FUNCTION_BLOCK FB_HighVoltTray EXTENDS FB_ActiveTarget

VAR
	//Hardware-Verküpfung
	pHighVoltSupplyRef	: POINTER TO FB_HighVoltSupply;
	
	//Prozessdaten
	nVoltageActual		: DINT;
	nCurrentActual		: DINT;	//in 10tel µA (10 enstpr. 1.0µA)

	//Variablen allgemeine Statemachine
	
	bCurrentMonitoring		: BOOL;
	bPwrCutOffTriggered		: BOOL;

	//Spec-Properties
	nVoltageChannel			: USINT;
	nCurrentLimit			: UINT; 		//Strombegrenzung der HV-Quelle //in 10tel µA (10 enstpr. 1.0µA)
	
	nPowerCutOffThreshold	: UINT;			//Stromüberwachung (Automatisches Abschalten bei Erreichen) //in 10tel µA (10 enstpr. 1.0µA)
											//wenn "0" , dann wird nicht überwacht
	tPowerCutOffTime		: TIME; 		//wenn Strom für diese Zeit die Abschaltschwelle überschreitet, dann wird abgeschaltet
	
	//****************************************Aktionvariablen****************************************************
	
	//Action: "SetVoltage"
	nVoltageSetpoint	: USINT;
	
	//Action: "SetCurrent"
	nCurrentSetpoint	: USINT;
	
	//Action: "SwitchVoltage"
	bVoltageOn			: BOOL;
	
	timer : TON;	//Stromüberwachung
	
	
END_VAR

IF pHighVoltSupplyRef = 0 THEN
	RETURN;
END_IF

pFbSafety^.M_MesBoxOn();

//durch Notaus oder Unlock werden die Kanäle ausgeschalten und müssen in jedem Fall
//manuell durch SwitchVoltage wieder eingeschalten werden
IF NOT pHighVoltSupplyRef^.bHVPSAvailable THEN
	pHighVoltSupplyRef^.M_SwitchVoltage(1,FALSE);
	pHighVoltSupplyRef^.M_SwitchVoltage(2,FALSE);
END_IF

//Stromüberwachung
nCurrentActual := pHighVoltSupplyRef^.M_GetCurrent();
IF bCurrentMonitoring AND NOT bPwrCutOffTriggered THEN
	IF nCurrentActual >= nPowerCutOffThreshold THEN
		//Strom muss für eine vorgegebene Zeit die Abschaltschwelle erreicht haben.
		timer(IN:= TRUE, PT:= tPowerCutOffTime);
		IF timer.Q THEN
			timer(IN:= FALSE);
			bPwrCutOffTriggered := TRUE; 
			pHighVoltSupplyRef^.M_SwitchVoltage(1,FALSE);
			pHighVoltSupplyRef^.M_SwitchVoltage(2,FALSE);
			stError.POU := E_POU.POU_FB_HighVoltTray;
			stError.ErrorId := E_ErrorIdCmd.ERRORID_OverCurrentHighVoltTray;
			stError.ObjectId := nObjectID;
			fbErrorList.M_Add(stError);			
		END_IF
	ELSE
		timer(IN:= FALSE);
	END_IF
END_IF

//Prozessdaten aktualisieren
stProcessData.nObjId := nObjectID;
stProcessData.n32Data[0] := BOOL_TO_DINT(bIsInit);
stProcessData.n32Data[1] := eCurrentState;
stProcessData.n32Data[2] := stError.ErrorId;

IF nVoltageChannel = 1 THEN
	stProcessData.n32Data[3] := BOOL_TO_DINT(NOT pHighVoltSupplyRef^.bDigiOutVoltage1);
ELSIF nVoltageChannel = 2 THEN
	stProcessData.n32Data[3] := BOOL_TO_DINT(NOT pHighVoltSupplyRef^.bDigiOutVoltage2);
END_IF

nVoltageActual := pHighVoltSupplyRef^.M_GetVoltage();
stProcessData.n32Data[4] := nVoltageActual;
stProcessData.n32Data[5] := nCurrentActual;

aObjProcData[nNotifyId] := stProcessData;

METHOD FB_init : BOOL
VAR_INPUT
	bInitRetains : BOOL; // if TRUE, the retain variables are initialized (warm start / cold start)
	bInCopyCode : BOOL;  // if TRUE, the instance afterwards gets moved into the copy code (online change)
END_VAR
eObjectType := E_ObjectType.OBJECTTYPE_HighVoltTray;
eObjectGroup := E_ObjectGroup.OBJECTGROUP_Target OR E_ObjectGroup.OBJECTGROUP_Device;
END_METHOD

METHOD M_CheckProcDataType : BOOL
VAR_INPUT
	eProcDataType : E_ProcDataType;
END_VAR
IF eProcDataType = E_ProcDataType.PROCDATATYPE_Voltage1 OR eProcDataType = E_ProcDataType.PROCDATATYPE_Current1 THEN
	M_CheckProcDataType := TRUE;
END_IF
END_METHOD

METHOD M_CurrentMonitoring
VAR_INPUT
	bOn : BOOL;
END_VAR
IF bOn THEN
	IF nPowerCutOffThreshold > 0 THEN
		bCurrentMonitoring := TRUE;		
	END_IF
ELSE
	bCurrentMonitoring := FALSE;
 	bPwrCutOffTriggered := FALSE;
END_IF
END_METHOD

METHOD M_ExeAction : ERRORID
VAR_INPUT
	refActionData	: REFERENCE TO ST_ActionData;	
END_VAR
CASE refActionData.eAction OF
	E_Action.ACTION_Init:
		bIsInit := TRUE;
		RETURN;
	E_Action.ACTION_SetVoltage:
		IF 	pHighVoltSupplyRef > 0 THEN
			pHighVoltSupplyRef^.M_SetVoltage(DINT_TO_INT(refActionData.aParams[1]));
			pHighVoltSupplyRef^.M_SetCurrent(nCurrentLimit);
		END_IF
	E_Action.ACTION_SwitchVoltage:
		IF 	pHighVoltSupplyRef > 0 THEN
			IF pHighVoltSupplyRef^.bHVPSAvailable THEN
				pHighVoltSupplyRef^.M_SwitchVoltage(nVoltageChannel,DINT_TO_BOOL(refActionData.aParams[1]));
			ELSE
				M_ExeAction := E_ErrorIdCmd.ERRORID_HighVoltSupplyOff;
			END_IF
		ELSE
			M_ExeAction := E_ErrorIdObjMgmt.ERRORID_InvalidHardwareRef;
		END_IF
	ELSE
		M_ExeAction := E_ErrorIdCmd.ERRORID_InvalidAction;	
END_CASE
END_METHOD

METHOD M_GetActionBusy : BOOL
VAR_INPUT
	eAction : E_Action;
END_VAR
IF eAction = eCurrentAction THEN
	M_GetActionBusy := TRUE;
END_IF
END_METHOD

METHOD M_GetAllProps : ERRORID
VAR_INPUT
	refCmdData : REFERENCE TO  ST_CmdData;
END_VAR
SUPER^.M_GetAllProps(refCmdData);
nCurrentPropIndex := nCurrentPropIndex + 1;
refCmdData.n32Data[nCurrentPropIndex] := nVoltageChannel;
nCurrentPropIndex := nCurrentPropIndex + 1;
refCmdData.n32Data[nCurrentPropIndex] := nCurrentLimit;
nCurrentPropIndex := nCurrentPropIndex + 1;
refCmdData.n32Data[nCurrentPropIndex] := nPowerCutOffThreshold;
nCurrentPropIndex := nCurrentPropIndex + 1;
refCmdData.n32Data[nCurrentPropIndex] := TIME_TO_DINT(tPowerCutOffTime);
END_METHOD

METHOD M_GetProcData : DINT
VAR_INPUT
	eProcDataType : E_ProcDataType;
END_VAR
IF eProcDataType = E_ProcDataType.PROCDATATYPE_Voltage1 THEN
	M_GetProcData := pHighVoltSupplyRef^.M_GetVoltage();
ELSIF eProcDataType = E_ProcDataType.PROCDATATYPE_Current1 THEN
	M_GetProcData := pHighVoltSupplyRef^.M_GetCurrent();
END_IF
END_METHOD

METHOD M_Reset
bBusy := TRUE;
eCurrentState := E_MachineState.MACHINESTATE_Reset;
M_CurrentMonitoring(FALSE);
END_METHOD

METHOD M_SetAllProps : ERRORID
VAR_INPUT
	refCmdData : REFERENCE TO  ST_CmdData;
END_VAR
M_SetAllProps := SUPER^.M_SetAllProps(refCmdData);

IF M_SetAllProps > 0 THEN
	RETURN;
END_IF

{IF defined (variable:fbHighVoltSupplyRef)}
pHighVoltSupplyRef := ADR(fbHighVoltSupplyRef);
{ELSE}
{warning 'implement errorId}
M_SetAllProps := E_ErrorIdObjMgmt.ERRORID_InvalidHardwareRef;
{END_IF}
nCurrentPropIndex := nCurrentPropIndex + 1;
nSpecPropIndex := nCurrentPropIndex;
IF refCmdData.n32Data[nCurrentPropIndex] >= 1 AND refCmdData.n32Data[nCurrentPropIndex] <= 2 THEN
	nVoltageChannel := DINT_TO_USINT(refCmdData.n32Data[nCurrentPropIndex]);
ELSE
	M_SetAllProps := E_ErrorIdObjMgmt.ERRORID_InvalidHardwareRef;
END_IF

nCurrentPropIndex := nCurrentPropIndex + 1;
nCurrentLimit := DINT_TO_UINT(refCmdData.n32Data[nCurrentPropIndex]);
nCurrentPropIndex := nCurrentPropIndex + 1;
nPowerCutOffThreshold := DINT_TO_UINT(refCmdData.n32Data[nCurrentPropIndex]);
nCurrentPropIndex := nCurrentPropIndex + 1;
tPowerCutOffTime := DINT_TO_TIME(refCmdData.n32Data[nCurrentPropIndex]);

nNoOfProps := nCurrentPropIndex + 1;
END_METHOD

METHOD M_SetSingleProp : ERRORID
VAR_INPUT
	refCmdData : REFERENCE TO  ST_CmdData;
END_VAR
IF nSpecPropIndex = refCmdData.aHeader[1] THEN
	IF refCmdData.n32Data[0] >= 1 OR refCmdData.n32Data[0] <= 2 THEN
		IF refCmdData.n32Data[0] <> nVoltageChannel THEN
			IF pHighVoltSupplyRef > 0 THEN
				pHighVoltSupplyRef^.M_SwitchVoltage(1,FALSE);
				pHighVoltSupplyRef^.M_SwitchVoltage(2,FALSE); 
			END_IF
			nVoltageChannel := DINT_TO_USINT(refCmdData.n32Data[0]);
		END_IF
	ELSE
		M_SetSingleProp := E_ErrorIdCmd.ERRORID_InvalidVoltageChannel;	
	END_IF
ELSIF (nSpecPropIndex + 1) = refCmdData.aHeader[1] THEN
	nCurrentLimit := DINT_TO_UINT(refCmdData.n32Data[0]);
	IF pHighVoltSupplyRef > 0 THEN
		pHighVoltSupplyRef^.M_SetCurrent(nCurrentLimit);
	END_IF
ELSIF (nSpecPropIndex + 2) = refCmdData.aHeader[1] THEN
	nPowerCutOffThreshold := DINT_TO_UINT(refCmdData.n32Data[0]);
ELSIF (nSpecPropIndex + 3) = refCmdData.aHeader[1] THEN
	tPowerCutOffTime := DINT_TO_TIME(refCmdData.n32Data[0]);
ELSE
	M_SetSingleProp := SUPER^.M_SetSingleProp(refCmdData);
END_IF
END_METHOD

PROPERTY P_bBusy : BOOL
GET
P_bBusy := bBusy;
END_GET
END_PROPERTY

PROPERTY P_bCanceled : BOOL
GET
P_bCanceled := bCanceled;
END_GET
END_PROPERTY

PROPERTY P_bError : BOOL
GET
IF eCurrentState = E_MachineState.MACHINESTATE_Error THEN
	P_bError := TRUE;
END_IF
END_GET
END_PROPERTY

PROPERTY P_bIsInit : BOOL
GET
P_bIsInit := bIsInit;
END_GET
SET
bIsInit := P_bIsInit;
END_SET
END_PROPERTY

PROPERTY P_bPwrCutOffTriggered : BOOL
GET
P_bPwrCutOffTriggered := bPwrCutOffTriggered;
END_GET
END_PROPERTY

PROPERTY P_bStopAllOnError : BOOL
GET
END_GET
END_PROPERTY

PROPERTY P_nCurrentVoltage : DINT
GET
P_nCurrentVoltage := nVoltageActual;
END_GET
END_PROPERTY

PROPERTY P_stError : ST_Error
GET
END_GET
END_PROPERTY

END_FUNCTION_BLOCK

(* stored: Version 1.1.0.1, ProductVersion 3.1.4022.18
   POU FB_HighVoltTray: Id {b14411df-784d-467c-989f-33a7aee080bd}, SpecialFunc None
   Method FB_init: Id {186bcc17-cfd2-444f-ba68-0a154951dd79}
   Method M_CheckProcDataType: Id {a3ed9780-b535-4d3e-a5b9-77710fdce5f7}
   Method M_CurrentMonitoring: Id {f9d38355-0248-49f8-9ae6-19668272f307}
   Method M_ExeAction: Id {0126e16c-e3bb-4e8f-95d7-0509df56c85f}
   Method M_GetActionBusy: Id {bb0c56a8-3a6b-4ac8-be7c-1caf0a366737}
   Method M_GetAllProps: Id {c58d8807-36e7-495b-95d6-135ba5f847a1}
   Method M_GetProcData: Id {11ff710c-ea16-4957-9c15-412b0ff47283}
   Method M_Reset: Id {892c5a7d-75ac-4c3c-aa85-0804e9898739}
   Method M_SetAllProps: Id {a17c4f64-c560-43e8-955f-f9432d728443}
   Method M_SetSingleProp: Id {7acf8738-3593-473e-ab93-c696c2fcd1f8}
   Property P_bBusy: Id {d6b3abc7-9e08-43d3-8835-10ad8c2c8332}
   Get Get: Id {f90adaf2-3e5e-4f1c-be2a-c0739b953d61}
   Property P_bCanceled: Id {ef22925e-d777-4203-8556-fe09d0971d2b}
   Get Get: Id {d035e83f-b3c0-4847-a6e3-7c513a64b9f8}
   Property P_bError: Id {62172918-b16e-4e6b-af88-22f5894ea239}
   Get Get: Id {90ba3ea7-be17-4ea6-be5f-9492d27b3929}
   Property P_bIsInit: Id {99c319b2-852d-4b75-9066-2fe403d7d514}
   Get Get: Id {d2cb6a9a-2a3a-45c6-8db9-722f03d3f2de}
   Set Set: Id {b0af8e08-f157-450d-851e-8fe261a41057}
   Property P_bPwrCutOffTriggered: Id {f4291e9f-d87b-4ebf-8923-b951b2f52192}
   Get Get: Id {8524ccca-a73c-4282-a2b7-81dbfb0de167}
   Property P_bStopAllOnError: Id {28da7f06-2236-46b7-b976-334e1966f0e3}
   Get Get: Id {c443913b-1438-4752-b1d8-9355777331e7}
   Property P_nCurrentVoltage: Id {23320105-96b0-423f-83f6-17b0f890c881}
   Get Get: Id {e2a1ddd3-0d6b-4eed-8f54-7c20df20f59e}
   Property P_stError: Id {955f92e7-6195-4cfd-bfbc-218c8256f34a}
   Get Get: Id {7c2f1c23-e449-46d8-a2c9-b4b6903d9b4f} *)
